FUNCTION_BLOCK SUBL_8_SETUP (* 8-variable local group subscriber for setup resource *)
  (* Standard: 61499-2 *)
  (* Version 1.0, 13-04-12, GASR, Universidade do Estado de Santa Catarina *)
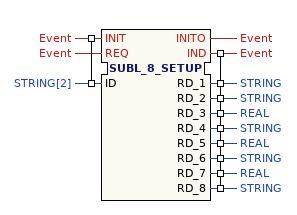
  EVENT_INPUT
    INIT WITH ID; (* Service Initialization *)
    REQ; (* Service Request *)
  END_EVENT
  EVENT_OUTPUT
    INITO; (* Initialization Confirm *)
    IND WITH RD_1, RD_2, RD_3, RD_4, RD_5, RD_6, RD_7, RD_8; (* Service Confirmation *)
  END_EVENT
  VAR_INPUT
    ID : ARRAY [0..1] OF STRING; (* Default id is the FB instance name *)
  END_VAR
  VAR_OUTPUT
    RD_1 : STRING; (* workplan.its_setup.its_origin.name *)
    RD_2 : STRING; (* workplan.its_setup.its_origin.location.name *)
    RD_3 : REAL; (* workplan.its_setup.its_origin.location.coordinates *)
    RD_4 : STRING; (* workplan.its_setup.its_origin.axis.its_id *)
    RD_5 : REAL; (* workplan.its_setup.its_origin.axis.direction_ratios *)
    RD_6 : STRING; (* workplan.its_setup.its_origin.ref_direction.its_id *)
    RD_7 : REAL; (* workplan.its_setup.its_origin.ref_direction_ratios *)
    RD_8 : STRING; (* current_tool *)
  END_VAR
  SERVICE SUBL_8_SETUP/PUBL_8_SETUP (* Data publication service *)
    SEQUENCE normal_establishment
      SUBL_8_SETUP.INIT(ID) -> PUBL_8_SETUP.INITO();
      PUBL_8_SETUP.INIT(ID) -> PUBL_8_SETUP.INITO();
    END_SEQUENCE
    SEQUENCE normal_data_transfer
      SUBL_8_SETUP.REQ(RD_1,RD_2,RD_3,RD_4,RD_5,RD_6,RD_7,RD_8) -> PUBL_8_SETUP.IND(SD_1,SD_2,SD_3,SD_4,SD_5,SD_6,SD_7,SD_8) -> SUBL_8_SETUP.CNF();
    END_SEQUENCE
  END_SERVICE
END_FUNCTION_BLOCK
